// TIA Portal project "Ejercicio2-Semaforo-TIA" (V14)

(* hardware
DEVICE "S7-1200 station_1"  S7-1200 Station
   slot 0: "Rack_0"  S7-1200 Rack  Rack  V1.0
   slot 1: "PLC_1"  CPU 1214C DC/DC/DC  6ES7 214-1AG40-0XB0  V4.2
*)

// ===== PLC "PLC_1"  CPU 1214C DC/DC/DC =====

VAR_GLOBAL   // PLC tag table "Tabla de variables estándar"
   "Clock_Byte" AT %MB0 : Byte;
   "Clock_10Hz" AT %M0.3 : Bool;
   "Clock_5Hz" AT %M0.1 : Bool;
   "Clock_2.5Hz" AT %M0.2 : Bool;
   "Clock_2Hz" AT %M0.3 : Bool;
   "Clock_1.25Hz" AT %M0.4 : Bool;
   "Clock_1Hz" AT %M0.5 : Bool;
   "Clock_0.625Hz" AT %M0.6 : Bool;
   "Clock_0.5Hz" AT %M0.7 : Bool;
   "System_Byte" AT %MB1 : Byte;
   "FirstScan" AT %M1.0 : Bool;
   "DiagStatusUpdate" AT %M1.1 : Bool;
   "AlwaysTRUE" AT %M1.2 : Bool;
   "AlwaysFALSE" AT %M1.3 : Bool;
   "LedVerde" AT %Q0.0 : Bool;
   "LedAmarillo" AT %Q0.1 : Bool;
   "LedRojo" AT %Q0.2 : Bool;
   "Encender" AT %I0.0 : Bool;
   "Marca" AT %M2.0 : Bool;
   "Tag_1" AT %MD100 : Time;
END_VAR

// folder: System blocks/Program resources

DATA_BLOCK "Verde"   // DB2
{ S7_Optimized_Access := 'TRUE' }
AUTHOR : Simatic
FAMILY : IEC
NAME : IEC_TMR
VERSION : 1.0
// stored: InstanceOfName IEC_TIMER
"IEC_TIMER"
BEGIN
END_DATA_BLOCK

DATA_BLOCK "Amarillo"   // DB3
{ S7_Optimized_Access := 'TRUE' }
AUTHOR : Simatic
FAMILY : IEC
NAME : IEC_TMR
VERSION : 1.0
// stored: InstanceOfName IEC_TIMER
"IEC_TIMER"
BEGIN
END_DATA_BLOCK

DATA_BLOCK "ROJO"   // DB5
{ S7_Optimized_Access := 'TRUE' }
AUTHOR : Simatic
FAMILY : IEC
NAME : IEC_TMR
VERSION : 1.0
// stored: InstanceOfName IEC_TIMER
"IEC_TIMER"
BEGIN
END_DATA_BLOCK

// folder: (top level)

FUNCTION "Semaforo" : Void   // FC2, LAD
TITLE = Bloque de Funcion Semaforo
{ S7_Optimized_Access := 'TRUE' }
VERSION : 0.1
   VAR_TEMP   // added for the SCL form of the ladder/FBD networks
      _w1 : Bool;
   END_VAR
BEGIN

REGION Network 1: Secuencia
   // Realizamos la secuencia del semaforo, al darle al pulsador encender, enciende el Temporizador "Verde" durante 20s, al terminar de contar, la señal Verde.Q normalmente abierta conmuta, obligando al Temporizador TOF "Amarillo".  En amarillo almacenamos en el indice MD100 de nombre Tag_1 para compararlo a la salida Q del temporizador. Si el valor almacenado del tipo Time es menor a T# 3s, el LedAmarillo permanecera prendido constantemente, si el valor almacenado es mayor, el LedAmarillo titilara con una frecuencia de 2Hz. Cumplido los 5s, el contacto NA del temporizador "Amarillo", que se encontraba cerrado, se abre, dandole asi, la señal al Temporizador "ROJO" para que realice su conteo, una vez que termina, se reinicia el ciclo.
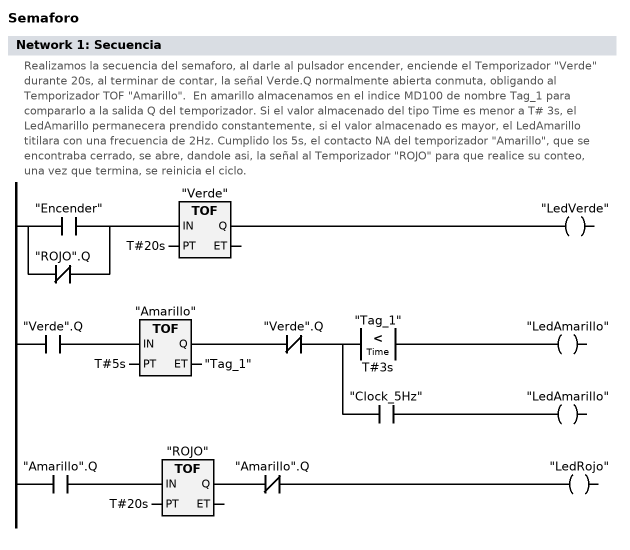
   "Verde".TOF(IN := "Encender" OR NOT "ROJO".Q, PT := T#20s);
   "LedVerde" := "Verde".Q;
   "Amarillo".TOF(IN := "Verde".Q, PT := T#5s, ET => "Tag_1");
   #_w1 := "Amarillo".Q AND NOT "Verde".Q;
   "LedAmarillo" := #_w1 AND ("Tag_1" < T#3s);
   "LedAmarillo" := #_w1 AND "Clock_5Hz";
   "ROJO".TOF(IN := "Amarillo".Q, PT := T#20s);
   "LedRojo" := "ROJO".Q AND NOT "Amarillo".Q;
END_REGION
END_FUNCTION

ORGANIZATION_BLOCK "Main"   // OB1, LAD, ProgramCycle
TITLE = "Main Program Sweep (Cycle)"
{ S7_Optimized_Access := 'TRUE' }
VERSION : 0.1
   VAR_INPUT
      Initial_Call : Bool;   // Initial call of this OB
      Remanence : Bool;   // =True, if remanent data are available
   END_VAR
BEGIN

REGION Network 1
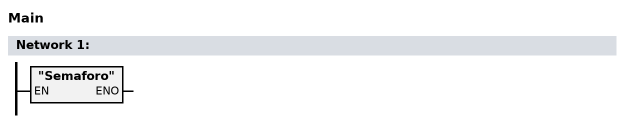
   RUNG wire#powerrail
      "Semaforo"()
   END_RUNG
   // the same network as SCL:
   "Semaforo"();
END_REGION
END_ORGANIZATION_BLOCK